TYPE ST_AXIS_SYNC_STATUS :
STRUCT
END_STRUCT
END_TYPE

(* stored: Version 1.1.0.1, ProductVersion 3.1.4024.11
   DUT ST_AXIS_SYNC_STATUS: Id {89c48860-cedc-45db-a099-2d8855b2948d} *)
